Fanuc KAREL source: NC0013.KL

-- PROVISIONAL review KL for V940-1; original PC SHA256 1a1a6fd3a53a1f177f3ec25195260d5e6e6dee429a14d2f7fd5752be27994281
-- Incomplete behavior may be omitted. Consult companion uncertainty JSON. Do not deploy.
PROGRAM NC0013
%NOLOCKGROUP
-- UNRESOLVED_LOCAL_POOL 1 cells at code offset 3; source declarations unknown
-- DIRECT_LOCAL_WORD_ACCESS alone does not prove INTEGER, REAL, or BOOLEAN
BEGIN
  -- V9_EXPOSED_INDEXED_TABLE_HINT layout=0001; 4 counted words exposed once; source arms/runtime held
  -- V9_CONDITION_STACK_HINT 2 bounded expression windows; static native code-base-relative target link; source arms held
  -- UNRESOLVED_PC offsets 0-8; opcodes 2B,2C,7B
  -- UNRESOLVED_PC offsets 13-20; opcodes 9D,23
  -- UNRESOLVED_PC offsets 25-38; opcodes 21,9D,57,79
  -- UNRESOLVED_PC offsets 43-61; opcodes 21,2E,52,23
  -- UNRESOLVED_PC offsets 66-71; opcodes 7A
  -- UNRESOLVED_PC offsets 76-89; opcodes 21,9D,57,79
  -- UNRESOLVED_PC offsets 94-112; opcodes 21,2E,52,23
  -- UNRESOLVED_PC offsets 117-122; opcodes 7A
  -- UNRESOLVED_PC offsets 127-141; opcodes 21,9D,52,23
  -- UNRESOLVED_PC offsets 156-160; opcodes 7F
  -- UNRESOLVED_PC offsets 165-169; opcodes 27,AA
  -- UNRESOLVED_PC offsets 174-178; opcodes 7F
END NC0013
